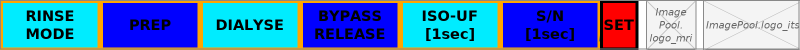
VISUALIZATION Header  // 800x50
    Rectangle (0,0 100x50), "RINSE MODE"
    Rectangle (100,0 100x50), "PREP"
    Rectangle (200,0 100x50), "DIALYSE"
    Rectangle (300,0 100x50), "BYPASS RELEASE", tooltip "BY PAS"
    Rectangle (400,0 100x50), "ISO-UF [1sec]"
    Rectangle (500,0 100x50), "S/N [1sec]"
    Image (600,0 25x50), image: ImagePool.logo_its
    Image (646,0 50x50), image: ImagePool.logo_mri
    Rectangle (600,0 38x50), "SET"
    Image (703,0 100x50), image: ImagePool.logo_its
END_VISUALIZATION

(* stored: Version 1.1.0.1, ProductVersion 3.1.4024.12
   Visu Header: Id {eed691dc-4eae-4ed1-a52b-032d96bbdb93} *)
